TYPE ST_Descriptor :
STRUCT
	stNames						: ST_Label;
	sUnit						: STRING(6);
	rValue						: REAL;
	rMin						: REAL;
	rMax						: REAL;
	rDefaultValue				: REAL;
	
END_STRUCT
END_TYPE

(* stored: Version 1.1.0.1
   DUT ST_Descriptor: Id {6599cd84-8a99-00ca-1312-c67e4a5fcf51} *)
